// TIA Portal V20 export
DATA_BLOCK "FSIDB_Main_Safety_RTG1"   // DB1, F_DB
NAME : FUSI
// stored: InstanceOfName FSFB_Main_Safety_RTG1, InstanceOfType FB
"FSFB_Main_Safety_RTG1"
   // VAR
   //    ESTOP : ESTOP1;
   // END_VAR
BEGIN
END_DATA_BLOCK
